//称重测试
PROGRAM LateBlanking_Weight_Test
VAR
	strBetryName: STRING;//文件名

    strBetryName2: STRING;//文件名
	bTest: BOOL;
	AA: UDINT;
	BB: UDINT;
	Weight_cese_1: Weight_cese;
	
	W_ton :Tc2_Standard.TON;
	

	
END_VAR



//称重平台上料
IF NOT Permit_Weigh AND NOT Weigh_Finish THEN
	Permit_WeighRack:=TRUE;
	ELSE
	Permit_WeighRack:=FALSE;
END_IF


W_ton(PT:=T#100MS);
Weight_date();


CASE weight_step OF 
0:
IF Permit_Weigh AND NOT Weigh_Finish AND NOT P3_Error[15]THEN
	weight_step:=10;
END_IF

10:
P3_Weight_gross.Weight_start:=TRUE;
W_ton.IN:=TRUE;
weight_step:=20;

20:
IF( P3_Weight_gross.Weight_finish  AND W_ton.Q)  OR  P3User2_Par.Shield[2]	THEN
	Permit_Weigh:=FALSE;
	Weigh_Finish:=TRUE;
	P3_Weight_gross.Weight_start:=FALSE;
	CellMemory[CellNo.Weight].Cell_weight:=P3_Weight_gross.bweight;
	CellMemory[CellNo.Weight].Weight:=1;
	weight_step:=30;
END_IF

30:
W_ton.IN:=FALSE;
P3_Weight_gross.Weight_finish:=FALSE;
weight_step:=0;
END_CASE






































(*IF bTest THEN
	
 STRING_TO_UTF8(pDstUTF8:=ADR(P3WeightSend.Data) , pSrcSTRING:=ADR(strBetryName) , nDstSize:=INT_TO_UINT( LEN(STR:=strBetryName )+1) );

 AA:=INT_TO_UDINT( LEN(STR:=strBetryName2 )+1);
  BB:=INT_TO_UDINT( LEN(STR:=strBetryName )+1);
 UTF8_TO_STRING(pDstSTRING:=ADR(strBetryName2) , pSrcUTF8:=ADR(P3WeightRec.Data) , nDstSize:=SIZEOF(P3WeightRec.Data) , nDstLen=> AA    );
 bTest:=FALSE;
END_IF*)

ACTION Weight_date:
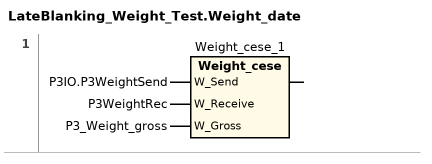
// NETWORK 1
Weight_cese_1(W_Send := P3IO.P3WeightSend, W_Receive := P3WeightRec, W_Gross := P3_Weight_gross); // Weight_cese
END_ACTION

END_PROGRAM

(* stored: Version 1.1.0.1, ProductVersion 3.1.4024.12
   POU LateBlanking_Weight_Test: Id {3b3f6510-c493-44c4-9436-171253fc6547}, SpecialFunc None
   Action Weight_date: Id {644be724-9cc3-4540-9374-34b8557baac3} *)
